Fanuc KAREL source: ko00134.KL

-- PROVISIONAL review KL for V1013-1; original PC SHA256 aa919a12ff5c3dc747738564a1139ff1aef44637c87525464bdc1e9e5e908bd9
-- Incomplete behavior may be omitted. Consult companion uncertainty JSON. Do not deploy.
PROGRAM KO00134
%NOLOCKGROUP
VAR
  R : REAL
  N : REAL
-- UNRESOLVED_DECL CFG type=00001c
-- UNRESOLVED_DECL OUT type=000102
BEGIN
  -- UNRESOLVED_PC offsets 5-13; opcodes 9D,64,23
  -- UNRESOLVED_PC offsets 18-29; opcodes 2E,23
  -- UNRESOLVED_PC offsets 34-44; opcodes 9D,22,A5
  -- UNRESOLVED_PC offsets 49-106; opcodes 27,22,22,22,22,22,22,22,76,7E,4A
  -- UNRESOLVED_PC offsets 111-115; opcodes 7F
END KO00134
